GLOBALCONSTANTS AID_IN (* Input number object attribute ids *)
  (* Standard: 61499-1; Description: Copyright (c) 2023 HR Agrartechnik GmbH This program and the accompanying materials are made available under the terms of the Eclipse Public License 2.0 which is available at https://www.eclipse.org/legal/epl-2.0/ SPDX-License-Identifier: EPL-2.0 *)
  (* Version 1.0, 2026-06-20, Franz Höpfinger, HR Agrartechnik GmbH *)
  PACKAGE isobus::UT::Q::const::AID;
  VAR_GLOBAL CONSTANT
    WIDTH : USINT := USINT#1; (* 1: AID_IN_WIDTH - Width in pixels. *)
    HEIGHT : USINT := USINT#2; (* 2: AID_IN_HEIGHT - Height in pixels. *)
    BACKGROUND_COLOUR : USINT := USINT#3; (* 3: AID_IN_BACKGROUND_COLOUR - Background colour index. *)
    FONT_ATT : USINT := USINT#4; (* 4: AID_IN_FONT_ATT - Object ID of a Font Attributes object. *)
    OPTIONS : USINT := USINT#5; (* 5: AID_IN_OPTIONS - Bitmask: Bit 0=Transparent, Bit 1=Display leading zeros, Bit 2=Display zero *)
    VARIABLE_REF : USINT := USINT#6; (* 6: AID_IN_VARIABLE_REF - Object ID of a Variable object. *)
    MIN_VALUE : USINT := USINT#7; (* 7: AID_IN_MIN_VALUE *)
    MAX_VALUE : USINT := USINT#8; (* 8: AID_IN_MAX_VALUE *)
    OFFSET : USINT := USINT#9; (* 9: AID_IN_OFFSET *)
    SCALE : USINT := USINT#10; (* 10: AID_IN_SCALE *)
    NUMB_DECIMALS : USINT := USINT#11; (* 11: AID_IN_NUMB_DECIMALS *)
    FORMAT : USINT := USINT#12; (* 12: AID_IN_FORMAT - Decimal display: 0 = fixed format decimal (####.nn), 1 = exponential format. *)
    JUSTIFICATION : USINT := USINT#13; (* 13: AID_IN_JUSTIFICATION - Justification: Bits 0-1 (Horizontal: 0=Left, 1=Middle, 2=Right), Bits *)
    VALUE : USINT := USINT#14; (* 14: AID_IN_VALUE - Current value. *)
    OPTIONS_2 : USINT := USINT#15; (* 15: AID_IN_OPTIONS_2 - Bitmask: Bit 0=Enabled, Bit 1=Real-time editing. *)
  END_VAR
END_GLOBALCONSTANTS
